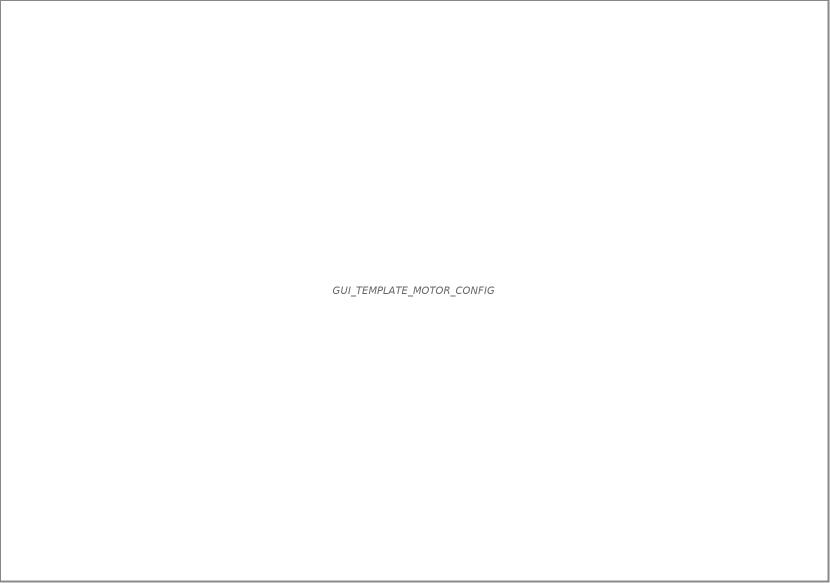
VISUALIZATION GUI_DROT_Cfg  // 830x583
    Frame (0,0 828x581)
        shows GUI_TEMPLATE_MOTOR_CONFIG(m_Instance := MAIN.drot.motor)
END_VISUALIZATION

(* stored: Version 1.1.0.1, ProductVersion 3.1.4022.12
   Visu GUI_DROT_Cfg: Id {ee7f9784-533d-4979-b33b-10fbafb23f56} *)
